(* CODESYS project SPT_Component_Base.library
   Company: Beckhoff Automation LLC
   DefaultNamespace: SPT_ComponentBase
   Version: 3.0.0
   Placeholder: SPT Component Base
   Title: SPT Component Base

Project tree, tasks and I/O mapping:
  libraries: SPT Base Types, * (Beckhoff Automation LLC); SPT Event Logger, * (Beckhoff Automation LLC); SPT PackML Base, * (Beckhoff Automation LLC); Tc2_Standard, * (Beckhoff Automation GmbH); Tc3_EventLogger, * (Beckhoff Automation GmbH); Tc3_Module, * (Beckhoff Automation GmbH); Tc3_System, * (Beckhoff Automation GmbH)
  DUT/
    data type ST_ComponentBase_Command
    data type ST_ComponentBase_Config
    data type ST_ComponentBase_HMI
    data type ST_ComponentBase_Status
  Function Blocks/
    function block FB_ComponentBase [ST]: AllowHMIControl, BlockHMIControl, Reset, CurrentAlarmSeverity, InSimulation, Name, ParentResponseDefinitions, CyclicLogic, CreateEvents, HMICommunication, Initialize, Monitoring, RaiseAlarm, RaiseAlarmWithStrings
  Interfaces/
    interface I_ComponentBase: AllowHMIControl, BlockHMIControl, Reset, CurrentAlarmSeverity, InSimulation, Name, ParentResponseDefinitions
  Project Information/
    function F_GetCompany [ST]
    function F_GetTitle [ST]
    function F_GetVersion [ST]
  Version/
    global variables Global_Version
  global variables Parameters_BaseComponent
*)

// DUT/ST_ComponentBase_Command
TYPE ST_ComponentBase_Command :
    STRUCT
        SimulatedOperation : BOOL;
        StandardOperation  : BOOL;
        Reset              : BOOL;
    END_STRUCT
END_TYPE

// DUT/ST_ComponentBase_Config
TYPE ST_ComponentBase_Config :
    STRUCT
        Name : STRING;
    END_STRUCT
END_TYPE

// DUT/ST_ComponentBase_HMI
TYPE ST_ComponentBase_HMI :
    STRUCT
        Config  : ST_ComponentBase_Config;
        Command : ST_ComponentBase_Command;
        Status  : ST_ComponentBase_Status;
    END_STRUCT
END_TYPE

// DUT/ST_ComponentBase_Status
TYPE ST_ComponentBase_Status :
    STRUCT
        InSimulation        : BOOL;
        Busy                : BOOL;
        Error               : BOOL;
        ErrorID             : UDINT;
        HMIControlAvailable : BOOL; //Set TRUE *FROM PLC* when HMI requests can be processed
    END_STRUCT
END_TYPE

// Version/Global_Version
{attribute 'TcGenerated'}
{attribute 'no-analysis'}
{attribute 'linkalways'}
// This function has been automatically generated from the project information.
VAR_GLOBAL CONSTANT
	{attribute 'const_non_replaced'}
	stLibVersion_SPT_Component_Base : ST_LibVersion := (iMajor := 3, iMinor := 0, iBuild := 0, iRevision := 0, nFlags := 1, sVersion := '3.0.0');
END_VAR

// Parameters_BaseComponent
{attribute 'qualified_only'}
VAR_GLOBAL CONSTANT
    COMPONENT_BASE_ALARM_COUNT : UDINT := 2;
END_VAR

// Function Blocks/FB_ComponentBase
//! @summary Basic framework of a component
FUNCTION_BLOCK ABSTRACT FB_ComponentBase EXTENDS FB_CyclicFB IMPLEMENTS I_ComponentBase
VAR
    //I_BasicComponent internal property variables
    _CurrentAlarmSeverity           : TcEventSeverity;
    _Name                           : STRING; //String name of the component
    _ParentFaultResponseDefinitions : ARRAY[0..4] OF E_AlarmResponse
        := [E_AlarmResponse.NoResponse, E_AlarmResponse.NoResponse, E_AlarmResponse.NoResponse, E_AlarmResponse.Abort_ImmediateError, E_AlarmResponse.Abort_ImmediateError];
    _Simulate : BOOL; //TRUE disables all hardware I/O and simulates input and output behavior

    //Alarming
    ComponentBaseAlarms : ARRAY[1..Parameters_BaseComponent.COMPONENT_BASE_ALARM_COUNT] OF FB_TcAlarm;

    //HMI Monitoring and control structure
    ComponentBase_HMI           : ST_ComponentBase_HMI;
    HMICommand_RT               : R_TRIG;
    HMICommandActive_Base       : BOOL;
    HMICommandActive_Descendant : BOOL;
END_VAR

//! @summary Sets permissive bit to allow HMI control of component functions
METHOD PUBLIC AllowHMIControl

//! @description This method is called as required by the parent module of this component
ComponentBase_HMI.Status.HMIControlAvailable := TRUE;
END_METHOD

//! @summary Clears permissive bit to allow HMI control of component functions
METHOD PUBLIC BlockHMIControl

//! @description This method is called as required by the parent module of this component
ComponentBase_HMI.Status.HMIControlAvailable := FALSE;
END_METHOD

//! @summary Clears error flags and error IDs for this component
METHOD PUBLIC Reset : BOOL
//This may or may not be called depending on the component type 

//which derives FB_ComponentBase
F_ClearAllEventsInClass(ComponentBaseAlarms);
Reset := TRUE;
END_METHOD

//! @summary Returns the current alarm severity for this component
PROPERTY CurrentAlarmSeverity : TcEventSeverity
GET
CurrentAlarmSeverity := _CurrentAlarmSeverity;
END_GET
END_PROPERTY

//! @summary Enable/Disable simulation logic for this component
PROPERTY InSimulation : BOOL
GET
InSimulation := _Simulate;
END_GET
SET
_Simulate := InSimulation;
END_SET
END_PROPERTY

//! @summary Get/Set this component's name
PROPERTY Name : STRING
GET
Name := _Name;
END_GET
SET
_Name := Name;
END_SET
END_PROPERTY

PROPERTY ParentResponseDefinitions : ARRAY[0..4] OF E_AlarmResponse
GET
ParentResponseDefinitions[TcEventSeverity.Verbose]  := _ParentFaultResponseDefinitions[TcEventSeverity.Verbose];
ParentResponseDefinitions[TcEventSeverity.Info]     := _ParentFaultResponseDefinitions[TcEventSeverity.Info];
ParentResponseDefinitions[TcEventSeverity.Warning]  := _ParentFaultResponseDefinitions[TcEventSeverity.Warning];
ParentResponseDefinitions[TcEventSeverity.Error]    := _ParentFaultResponseDefinitions[TcEventSeverity.Error];
ParentResponseDefinitions[TcEventSeverity.Critical] := _ParentFaultResponseDefinitions[TcEventSeverity.Critical];
END_GET
SET
_ParentFaultResponseDefinitions[TcEventSeverity.Verbose]  := ParentResponseDefinitions[TcEventSeverity.Verbose];
_ParentFaultResponseDefinitions[TcEventSeverity.Info]     := ParentResponseDefinitions[TcEventSeverity.Info];
_ParentFaultResponseDefinitions[TcEventSeverity.Warning]  := ParentResponseDefinitions[TcEventSeverity.Warning];
_ParentFaultResponseDefinitions[TcEventSeverity.Error]    := ParentResponseDefinitions[TcEventSeverity.Error];
_ParentFaultResponseDefinitions[TcEventSeverity.Critical] := ParentResponseDefinitions[TcEventSeverity.Critical];
END_SET
END_PROPERTY

//! @summary This method serves as the entry point for all underlying FB logic
METHOD PUBLIC CyclicLogic

//! @description This method should be called cyclically by descendant function blocks by invoking <c>SUPER^.CyclicLogic()</c>.  Alternatively, the contents of this method could be reimplemented entirely in which case a call to this method would not be necessary.
IF NOT _InitComplete THEN
    _InitComplete := Initialize();
    RETURN;
END_IF

Monitoring();       //Constant error and status monitoring
HMICommunication(); //Keeps the HMI data up to date, and processes requests from the HMI for this component
END_METHOD

//! @summary Initializes event function blocks using this components's name
{attribute 'call_after_online_change_slot' := '<slot>'}
METHOD PROTECTED CreateEvents

//! @description This method is called by <c>Initialize()</c> as required
F_CreateAllEventsInClass(Alarms     := ComponentBaseAlarms,
                         ClassSize  := SIZEOF(TC_EVENTS.ComponentBase),
                         pInitEvent := ADR(TC_EVENTS.ComponentBase.InitReferenceEvent),
                         Prefix     := _Name);
END_METHOD

//! @summary Provides interlocks for HMI control and updates HMI status information for this component
METHOD PROTECTED HMICommunication

//! @description This method is called cyclically by <c>CyclicLogic()</c>
//Extend this method in extended FBs to communicate specific implementation data

//Process HMI requests
HMICommand_RT(CLK := (ComponentBase_HMI.Status.HMIControlAvailable AND NOT HMICommandActive_Descendant) AND
                     (ComponentBase_HMI.Command.Reset XOR ComponentBase_HMI.Command.SimulatedOperation XOR ComponentBase_HMI.Command.StandardOperation));

//Desendant components should observe this to interlock HMI commands
HMICommandActive_Base :=
    ComponentBase_HMI.Status.HMIControlAvailable AND (ComponentBase_HMI.Command.Reset OR ComponentBase_HMI.Command.SimulatedOperation OR ComponentBase_HMI.Command.StandardOperation);

IF HMICommand_RT.Q THEN
    IF ComponentBase_HMI.Command.Reset THEN
        Reset();
    END_IF

    IF ComponentBase_HMI.Command.SimulatedOperation THEN
        _Simulate := TRUE;
    END_IF

    IF ComponentBase_HMI.Command.StandardOperation THEN
        _Simulate := FALSE;
    END_IF
END_IF

//Update HMI status info
ComponentBase_HMI.Config.Name         := _Name;
ComponentBase_HMI.Status.Busy         := _Busy;
ComponentBase_HMI.Status.Error        := _Error;
ComponentBase_HMI.Status.InSimulation := _Simulate;
ComponentBase_HMI.Status.ErrorID      := _ErrorID;
END_METHOD

//! @summary Basic component initialization logic
METHOD PROTECTED Initialize : BOOL;

//! @description This method is called by <c>CyclicLogic()</c> as required
//Extend initialize as needed in extended FBs
CreateEvents();
Initialize := TRUE;
END_METHOD

//! Provides basic error detection and event handling for this component
METHOD PROTECTED Monitoring

(*! @descriptionThis method is called cyclically by <c>CyclicLogic()</c>*)
//Extend from extended FB with monitoring logic
IF NOT ComponentBaseAlarms[E_ComponentBase.SimulationWarning].bRaised AND _Simulate THEN
    ComponentBaseAlarms[E_ComponentBase.SimulationWarning].Raise(0);
ELSIF ComponentBaseAlarms[E_ComponentBase.SimulationWarning].bRaised AND NOT _Simulate THEN
    ComponentBaseAlarms[E_ComponentBase.SimulationWarning].Clear(0, 0);
END_IF

_CurrentAlarmSeverity := TcEventSeverity.Verbose;
_CurrentAlarmSeverity := F_GetMaxSeverityRaised(Alarms := ComponentBaseAlarms, CurrentSeverity := _CurrentAlarmSeverity);
END_METHOD

//! @summary Raise an alarm, passing the faulted FB's error ID as a paramter
METHOD PROTECTED RaiseAlarm
VAR_IN_OUT
    Alarm : FB_TcAlarm;
END_VAR
F_RaiseAlarm(Alarm := Alarm);
END_METHOD

//! @summary Raises an alarm and passes string arguments as parameters for extra fault context/info
METHOD PROTECTED RaiseAlarmWithStrings
VAR_IN_OUT
    Alarm : FB_TcAlarm; //! Alarm to be raised
END_VAR

VAR_INPUT
    String_1 : STRING; //! First string parameter (The Name of this component will be applied first automatically)
    String_2 : STRING; //! Second string parameter
END_VAR
F_RaiseAlarmWithStringsAndFlags(Alarm     := Alarm,
                                ErrorFlag := _Error,
                                ErrorID   := _ErrorID,
                                String_1  := _Name,
                                String_2  := String_1,
                                String_3  := String_2);
END_METHOD

END_FUNCTION_BLOCK

// Interfaces/I_ComponentBase
INTERFACE I_ComponentBase EXTENDS I_CyclicFB

METHOD PUBLIC AllowHMIControl
VAR_INPUT
END_VAR
END_METHOD

METHOD PUBLIC BlockHMIControl
VAR_INPUT
END_VAR
END_METHOD

METHOD PUBLIC Reset : BOOL
END_METHOD

PROPERTY CurrentAlarmSeverity : TcEventSeverity
GET
END_GET
END_PROPERTY

PROPERTY InSimulation : BOOL
GET
END_GET
SET
END_SET
END_PROPERTY

PROPERTY Name : STRING
GET
END_GET
SET
END_SET
END_PROPERTY

PROPERTY ParentResponseDefinitions : ARRAY[0..4] OF E_AlarmResponse
GET
END_GET
SET
END_SET
END_PROPERTY

END_INTERFACE

// Project Information/F_GetCompany
// This function has been automatically generated from the project information.
{attribute 'signature_flag' := '1073741824'}
{attribute 'TcGenerated'}
{attribute 'no-analysis'}
FUNCTION F_GetCompany : WSTRING
VAR_INPUT
	
END_VAR

F_GetCompany := "Beckhoff Automation LLC";

END_FUNCTION

// Project Information/F_GetTitle
// This function has been automatically generated from the project information.
{attribute 'signature_flag' := '1073741824'}
{attribute 'TcGenerated'}
{attribute 'no-analysis'}
FUNCTION F_GetTitle : WSTRING
VAR_INPUT
	
END_VAR

F_GetTitle := "SPT Component Base";

END_FUNCTION

// Project Information/F_GetVersion
// This function has been automatically generated from the project information.
{attribute 'signature_flag' := '1073741824'}
{attribute 'TcGenerated'}
{attribute 'no-analysis'}
FUNCTION F_GetVersion : ST_LibVersion
VAR_INPUT
	
END_VAR

F_GetVersion.iMajor := 3;
F_GetVersion.iMinor := 0;
F_GetVersion.iBuild := 0;
F_GetVersion.iRevision := 0;
F_GetVersion.sVersion := '3.0.0';
F_GetVersion.nFlags := 1;

END_FUNCTION
